// TIA Portal V20 export
DATA_BLOCK "InstInterfaceSignalsConv_BA40"   // DB136
// stored: InstanceOfName CallInterfaceSignalsConv, InstanceOfType FB
"CallInterfaceSignalsConv"
   // VAR_INPUT
   //    InterfaceTestMode : Bool;
   // END_VAR
   // VAR_OUTPUT
   //    signalsR2S : "typeReelCutToStack";
   //    signalsS2R : "typeStackToReelCut";
   // END_VAR
   // VAR_IN_OUT
   //    CommR2S : Array[0..95] of Bool;
   //    CommS2R : Array[0..95] of Bool;
   //    InterfaceTestButton : "LER_SignalsInput";
   // END_VAR
   // VAR
   //    statWordBuffer_1 : Array[0..5] of Word;
   //    statWordBuffer_2 : Array[0..5] of Word;
   // END_VAR
BEGIN
END_DATA_BLOCK
